TYPE U_TRANSLATE_IN :
UNION
	nArray :	ARRAY[0..15] OF BYTE;
	Label :		S_NAMES_IN;
END_UNION
END_TYPE

(* stored: Version 1.1.0.1, ProductVersion 3.1.4024.6
   DUT U_TRANSLATE_IN: Id {a179c0df-6497-4103-9949-4d272c8f2db1} *)
